// TwinCAT 3 PLC project OCPPServer
// Title: TwinCAT IoT OCPP Server GettingStarted
// Company: Beckhoff Automation GmbH & Co. KG
// ProjectVersion: 1.0.3.0
// ProgramVersion: 3.1.4026.16
// libraries:
//   Tc2_Standard, * (Beckhoff Automation GmbH)
//   Tc2_System, * (Beckhoff Automation GmbH)
//   Tc3_OCPP, * (Beckhoff Automation GmbH)
// project tree:
//   DUTs/ ST_OCPP_BootNotification.TcDUT
//   / PlcTask.TcTTO
//   POUs/ MAIN.TcPOU
// (motion and I/O tree: see PLC project ocppclient)
// real-time tasks:
//   TASK PlcTask: cycle T#10ms, priority 20, ADS port 350
//   TASK PlcTask1: cycle T#10ms, priority 21, ADS port 351

CONFIGURATION OCPPServer
    RESOURCE PLC ON TwinCAT3
        TASK PlcTask(INTERVAL := T#10ms, PRIORITY := 21);
        PROGRAM MAIN WITH PlcTask : MAIN;
    END_RESOURCE
END_CONFIGURATION

// ---- DUTs/ST_OCPP_BootNotification.TcDUT
TYPE ST_OCPP_BootNotification :
STRUCT
	sModel 				: STRING(31);
	sVendor 			: STRING(31);
	sChargeBoxSerial 	: STRING(31);
	sChargePointSerial 	: STRING(31);
	sFirmwareVersion 	: STRING(63);
	sMeterSerial 		: STRING(31);
	sMeterType 			: STRING(31);
END_STRUCT
END_TYPE

// ---- POUs/MAIN.TcPOU
PROGRAM MAIN
VAR
	// Server param
	stServerParam 		: ST_OCPP1_ServerParam := (nPort:=8080,eAuthMode:=E_OCPP1_AuthenticationMode.None, eEncryptionMode := E_OCPP_EncryptionMode.None,eDebugLevel:=E_OCPP_DebugLevel.MessageLogFile, eTraceLevel:=TcTraceLevel.tlVerbose);
	fbOcppServer		: FB_OCPP1_Server(stServerParam);
	eAction 			: E_OCPP1_Action;
	hMessageId 			: T_OCPP_MessageId;
	hStationId			: UDINT;
	
	// Boot notification
	stBootNotification  : ST_OCPP_BootNotification;
	
	// Authorize
	sIdTag				: T_OCPP1_IdToken;
	
	// Transactions
	nConnectorId		: UDINT;
	nMeterStart			: UDINT;
	nMeterStop			: UDINT;
	nTimestamp			: ULINT;
	nTransactionId		: UDINT;
	nTransactionIdRecv	: UDINT;
	eReason				: E_OCPP1_Reason;
	
	// Status notification
	nConnectorIdStatus	: UDINT;
	eError				: E_OCPP1_ChargePointError;
	eStatus				: E_OCPP1_ChargePointStatus;
END_VAR

CASE eAction OF
	E_OCPP1_Action.None:
		IF NOT fbOcppServer.bError AND fbOcppServer.bValid THEN
			fbOcppServer.PollRequest(eAction => eAction, hMessageId => hMessageId, hStationId => hStationId);
		ELSE
			// Implement error handling here
		END_IF
	E_OCPP1_Action.BootNotification:
		IF fbOcppServer.RecvBootNotification(hStationId, hMessageId=>hMessageId, 			
			sModel				=> stBootNotification.sModel,
			sVendor				=> stBootNotification.sVendor,
			sChargeBoxSerial	=> stBootNotification.sChargeBoxSerial,
			sChargePointSerial	=> stBootNotification.sChargePointSerial,
			sFirmwareVersion	=> stBootNotification.sFirmwareVersion,
			sMeterSerial		=> stBootNotification.sMeterSerial,
			sMeterType			=> stBootNotification.sMeterType)
		THEN
			fbOcppServer.RespBootNotification(hStationId, hMessageId, E_OCPP1_RegistrationStatus.Accepted);
			eAction := E_OCPP1_Action.None;
		END_IF
	E_OCPP1_Action.Heartbeat:
		IF fbOcppServer.RecvHeartbeat(hMessageId => hMessageId, hStationId) THEN
			fbOcppServer.RespHeartbeat(hStationId:=hStationId,hMessageId:=hMessageId);
			eAction := E_OCPP1_Action.None;
		END_IF
	E_OCPP1_Action.Authorize:
		IF fbOcppServer.RecvAuthorize(hStationId, sIdTag => sIdTag, hMessageId => hMessageId) THEN
			IF sIdTag='Test123' THEN
				fbOcppServer.RespAuthorize(hStationId:=hStationId, hMessageId:=hMessageId, E_OCPP1_AuthorizationStatus.Accepted);
				eAction := E_OCPP1_Action.None;
			END_IF
		END_IF
	E_OCPP1_Action.StartTransaction:
		IF fbOcppServer.RecvStartTransaction(hStationId, hMessageId => hMessageId, sIdTag => sIdTag, nConnectorId => nConnectorId, nMeterStart => nMeterStart, nTimestamp => nTimestamp) THEN
			nTransactionId:=nTransactionId+1;
			fbOcppServer.RespStartTransaction(hStationId, hMessageId, E_OCPP1_AuthorizationStatus.Accepted, nTransactionId:=nTransactionId);
			eAction := E_OCPP1_Action.None;
		END_IF
	E_OCPP1_Action.StopTransaction:
		IF fbOcppServer.RecvStopTransaction(hStationId, hMessageId => hMessageId, sIdTag => sIdTag, nTransactionId => nTransactionIdRecv, nConnectorId => nConnectorId, nMeterStop => nMeterStop, nTimestamp => nTimestamp, eReason => eReason) THEN
			fbOcppServer.RespStopTransaction(hStationId, hMessageId, E_OCPP1_AuthorizationStatus.Accepted);
			eAction := E_OCPP1_Action.None;
		END_IF
	E_OCPP1_Action.StatusNotification:
		IF fbOcppServer.RecvStatusNotification(hStationId, hMessageId => hMessageId, nConnectorId => nConnectorIdStatus, eError => eError, eStatus => eStatus) THEN
			fbOcppServer.RespStatusNotification(hStationId, hMessageId);
			eAction := E_OCPP1_Action.None;
		END_IF
END_CASE

END_PROGRAM
